{attribute 'linkalways'} 
{attribute 'no_explicit_call' := 'This FB is a CLASS and must be accessed using methods or properties'}
{attribute 'enable_dynamic_creation'}
FUNCTION_BLOCK _DINT EXTENDS DatatypeBase
VAR
	localData : DINT;
	activeData : REFERENCE TO DINT REF= localData;
END_VAR

PROPERTY PUBLIC Address : PVOID
GET
Address := ADR(activeData);
END_GET
END_PROPERTY

METHOD PUBLIC ClearReference
VAR_INPUT
END_VAR
activeData REF= localData;
END_METHOD

METHOD PUBLIC Clone : I_Datatype
VAR
    pClone : POINTER TO _DINT;
END_VAR
pClone := __NEW(_DINT(InitialValue := Value));
Clone := pClone^;
END_METHOD

METHOD FB_init : BOOL
VAR_INPUT
	bInitRetains : BOOL; // if TRUE, the retain variables are initialized (warm start / cold start)
	bInCopyCode : BOOL;  // if TRUE, the instance afterwards gets moved into the copy code (online change)
	InitialValue : DINT;
END_VAR
localData := InitialValue;
END_METHOD

PROPERTY PUBLIC IecType : T_MAXSTRING
GET
IecType := 'DINT';
END_GET
END_PROPERTY

METHOD PUBLIC MakeReferenceTo
VAR_INPUT
	ReferenceTarget : REFERENCE TO DINT;
END_VAR
activeData REF= ReferenceTarget;
END_METHOD

METHOD PUBLIC SerializeWith
VAR_INPUT
	Serializer : I_Serializer;
END_VAR
Serializer.AddDint(activeData);
END_METHOD

PROPERTY PUBLIC Size : UDINT
GET
Size := SIZEOF(activeData);
END_GET
END_PROPERTY

METHOD TryDeserializeFrom : BOOL
VAR_INPUT
	Deserializer : I_Deserializer;
	Feedback : I_DeserializerFeedback;
END_VAR
TryDeserializeFrom := Deserializer.TryGetDint(activeData, Feedback);
END_METHOD

METHOD TryMakeReferenceTo : BOOL
VAR_INPUT
	Target : I_Datatype;
END_VAR
VAR
	pTargetData : POINTER TO DINT;
END_VAR
IF NOT (Target.IecType = IecType) THEN
	RETURN;
END_IF

pTargetData := Target.Address;
activeData REF= pTargetData^;
TryMakeReferenceTo := TRUE;
END_METHOD

PROPERTY PUBLIC Value : DINT
GET
Value := activeData;
END_GET
SET
activeData := Value;
END_SET
END_PROPERTY

END_FUNCTION_BLOCK

(* stored: Version 1.1.0.1, ProductVersion 3.1.4024.12
   POU _DINT: Id {65446692-a02d-4fc4-b466-67cb26841dd9}, SpecialFunc None
   Folder Constructor: Id {eac34c2d-e173-4410-9b00-5cc2d1621eb4}
   Property Address: Id {69925cc3-0822-482e-8d7e-caa88419cc92}
   Get Get: Id {8fd74165-734f-4ae5-87c5-01beae6051aa}
   Method ClearReference: Id {1f8d5e49-0476-4514-8c7b-ab50fc7d47b7}
   Method Clone: Id {ea3eb245-d34d-4c0d-8040-a829a54ac6b2}
   Method FB_init: Id {805990b5-1e2d-43ad-8631-4f839e012038}
   Property IecType: Id {4c117028-b45a-42c7-82ab-8ed0471c82fc}
   Get Get: Id {27304f57-6fd4-48d6-9f4e-7e6cbc2a82be}
   Method MakeReferenceTo: Id {6ed8112e-bd9f-47d8-93fc-f014f84e363b}
   Method SerializeWith: Id {6f27ee4d-0600-498a-a871-6687734f5d4d}
   Property Size: Id {2b4187e7-2b2e-4341-9414-e66a3d831fd3}
   Get Get: Id {db624b55-7b7e-4814-b3d8-5579388d26b3}
   Method TryDeserializeFrom: Id {4b8763a7-c048-4797-8818-d3d2131d4d4c}
   Method TryMakeReferenceTo: Id {bba1a4f3-2e9f-4afb-ad98-e91b315f70d0}
   Property Value: Id {95d8e7ae-8166-41ea-b32a-844f1aa026c3}
   Get Get: Id {2ec9e88b-3b61-4e4c-b452-442f721c777e}
   Set Set: Id {dd16e723-ba1a-41d9-bb2f-58f02121a75a} *)
